TEXTLIST TextList_Users_Menu
  1 = 'Gestion des utilisateurs\n' | FR: 'Gestion des utilisateurs' | EN: 'User management'
  2 = 'Identifiant' | FR: 'Identifiant' | EN: 'Login'
  17 = 'Save on disk' | FR: "Les groupes et utilisateurs\nvont être sauvegardés sur le disque.\nL'ancienne sauvegarde sera supprimée.\nConfirmer?" | EN: 'Users and groups will be \nsaved on disk. \nLast backup will be deleted. \nConfirm?'
  3 = 'Déconnexion' | FR: 'Confimez vous la déconnexion?' | EN: 'Confirm disconnection?'
  4 = 'Identification' | FR: 'Identification' | EN: 'Identification'
  5 = 'Login' | FR: 'Identifiant' | EN: 'Login'
  6 = 'Password' | FR: 'Mot de passe' | EN: 'Password'
  19 = 'Confirm supp groupe' | FR: 'Confirmer la suppression du groupe?' | EN: 'Confirm the group deletion?'
  18 = 'Confirm supp user' | FR: "Confirmer la suppression de l'utilisateur?" | EN: 'Confirm the user deletion?'
  21 = 'Confirm pwd' | FR: 'Confimation du mot de passe' | EN: 'Password confirmation'
  30 = 'Temps av deco' | FR: 'Temps avant déconnexion automatique :' | EN: 'Time before automatic logout:'
  31 = 'Deco auto utilisee' | FR: 'Utilisation de la déconnexion automatique :' | EN: 'Automatic logout used:'
  7 = 'user actu' | FR: 'Utilisateur actuel' | EN: 'Current user'
  8 = 'group actu' | FR: 'Groupe' | EN: 'Group'
  9 = 'Connexion' | FR: 'Connexion' | EN: 'Connection'
  10 = 'Déconnexion' | FR: 'Déconnexion' | EN: 'Disconnection'
  11 = 'droits par défaut' | FR: 'Droits\npar défaut' | EN: 'Rights\nby default'
  12 = 'Users' | FR: 'Utilisateurs' | EN: 'Users'
  13 = 'Groups' | FR: 'Groupes' | EN: 'Groups'
  14 = 'Charger' | FR: 'Charger' | EN: 'Load'
  15 = 'Sauvegarder' | FR: 'Sauvegarder' | EN: 'Save'
  16 = 'Options' | FR: 'Options' | EN: 'Options'
  20 = 'laod from disk' | FR: 'Les groupes et utilisateurs\nvont être restaurés depuis le disque\nLes groupes et utilisateurs actuels \nvont être écrasés. Confirmer?' | EN: 'Users and groups will be \nrestored from disk. \nCurrent groups and users will be deleted. \nConfirm?'
   = ''
END_TEXTLIST

(* stored: Version 1.1.0.1, ProductVersion 3.1.4024.10
   TextList TextList_Users_Menu: Id {7b9b9e61-464b-4b36-afdc-d1b0bd370a93} *)
